RoboDK station: arctos_demo.rdk

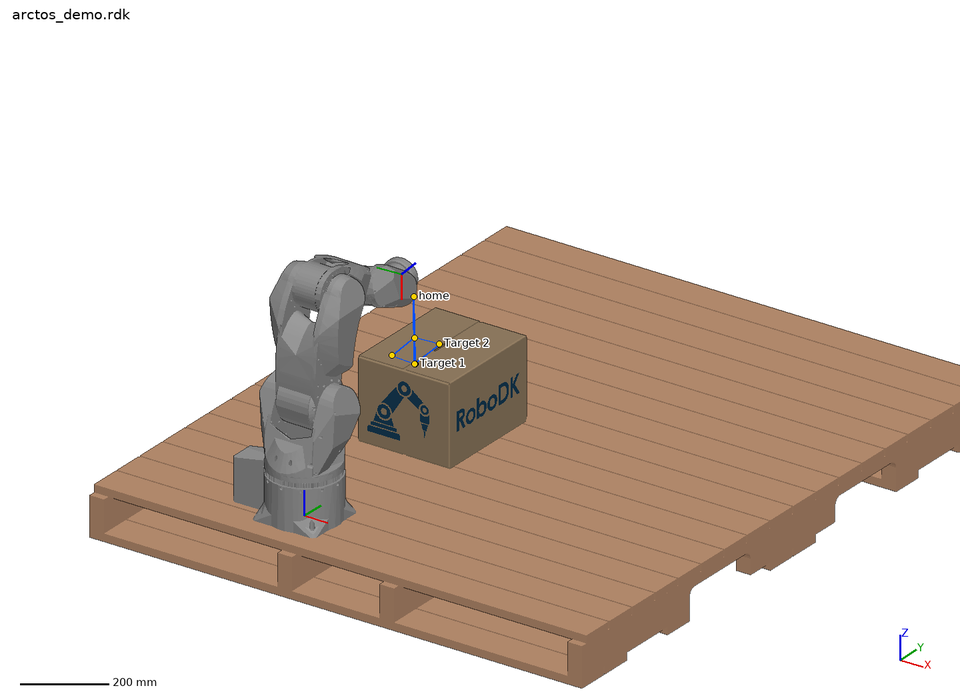
[picture v0: the station drawn from its stored meshes, robots at their saved joint values, targets as dots, program paths as lines]
Station arctos_demo (saved by RoboDK 6.0.1). Poses are relative to the parent item; angles as X-Y-Z fixed-axis rotations.
  - robot Arctos: 6 axes
      modified DH rows (alpha deg, a mm, theta deg, d mm): 0, 0, 0, 287.872; -90, 20.174, -90, 0; 0, 260.986, 0, 0; -90, 19.219, 0, 260.753; 90, 0, 0, 0; -90, 0, 180, 74.745
      joint limits [-200, -125, -50, -200, -100, -200] to [200, 75, 100, 200, 100, 200]; home [0, 0, 0, 0, 0, 0]; saved at [88.883, -9.103, -16.482, 12.937, -27.654, 11.654]
    - frame Arctos Base at (0, 0, 0) mm
    - tool Tool 1, TCP at (63, -17, 24.4) mm
  - object Pallet 1625x1350mm at (103.37, 1200.91, 945.52) mm, rotated rx -87.69 ry 84.94 rz 7.27 deg, size 1350 x 1650 x 125 mm, geometry from Pallet-1625x1350mm.sld
  - object Box 12x10in (Closed) at (-120, 380, 0) mm, size 252 x 305.4 x 216.7 mm, geometry from Box-12x10in-Closed.sld
  - frame Frame 2 at (0, 0, 0) mm
    - target Target 1 (Cartesian target) at (14.68, 411.52, 219.65) mm, rotated rx 0 ry 88.54 rz 94.85 deg; joints [88.843, -35.139, -26.856, 6.706, -63.62, 3.144] of Arctos
    - target Target 2 (Cartesian target) at (5.38, 521.09, 222.45) mm, rotated rx 0 ry 88.54 rz 94.85 deg; joints [90.416, -50.49, 5.427, 6.097, -46.69, 4.304] of Arctos
    - target Target 3 (Cartesian target) at (-59.39, 515.6, 222.45) mm, rotated rx 0 ry 88.54 rz 94.85 deg; joints [99.306, -50.492, 5.431, -6.128, -46.69, -4.326] of Arctos
    - target Target 4 (Cartesian target) at (-50.93, 415.99, 219.9) mm, rotated rx 0 ry 88.54 rz 94.85 deg; joints [100.698, -36.364, -24.213, -6.612, -62.203, -3.244] of Arctos
    - target Target 5 (Cartesian target) at (14, 411, 219.9) mm, rotated rx 0.01 ry 88.54 rz 94.86 deg; joints [88.967, -35.019, -26.999, 6.566, -63.636, 3.077] of Arctos
    - target home (Cartesian target) at (14.37, 406.68, 389.85) mm, rotated rx 0.01 ry 88.54 rz 94.86 deg; joints [88.883, -9.103, -16.482, 12.937, -27.654, 11.654] of Arctos
  - program 程序1 (13 instructions, listed below)
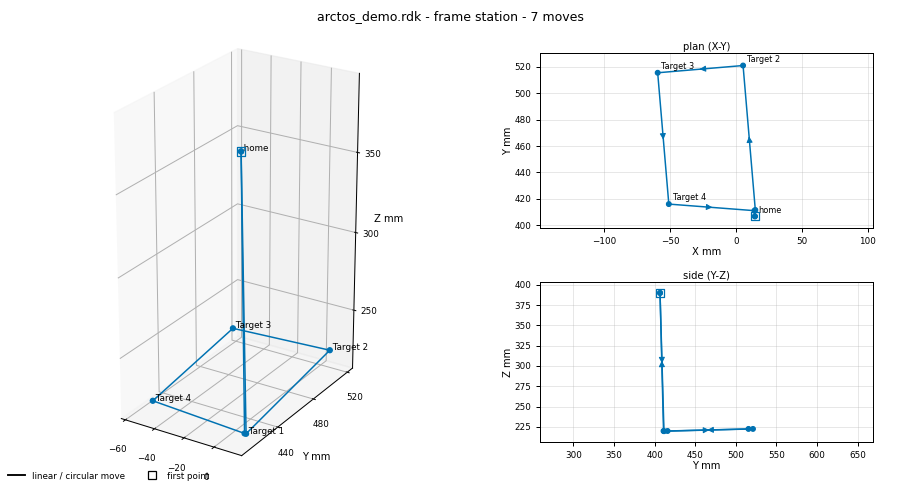
[picture p0: tool path of arctos_demo.rdk in frame station, 7 of 7 moves have a stored position in this frame; points joined in program order, loops and branches not executed]

--- program 程序1 (robot Arctos) ---
  设置参考: Frame 2
  设置工具: Tool 1
  MoveL (home)
  MoveL (Target 1)
  暂停 2.0 s
  Extruder(1)
  MoveL (Target 2)
  MoveL (Target 3)
  MoveL (Target 4)
  MoveL (Target 5)
  暂停 2.0 s
  Extruder(0)
  MoveL (home)
